FUNCTION Matrix_DeterminateSquare : BOOL
VAR_INPUT
	M : REFERENCE TO Matrix;
END_VAR
VAR_OUTPUT
	Res : LREAL;
END_VAR
VAR
	Sum : LREAL;
	Sign : LREAL;
	SubMatrix : ShrunkMatrixAccessor;
	
	Ci : UINT;
END_VAR

IF NOT(M.IsSquare) OR M.IsEmpty THEN
	Matrix_DeterminateSquare := FALSE;
	Res := 0;
	RETURN;
END_IF

Matrix_DeterminateSquare := TRUE;

IF M.Length = 1 THEN
	Res := M.GetRC(0,0);
ELSE
	Sum := 0;
	FOR Ci := 0 TO M.Cols-1 DO
		Sign := ((UINT_TO_INT(Ci)+1) MOD 2)*2 -1;//even columns are positive, odd columns are negative
		SubMatrix := M.GetShrunkMatrixAccessor(0,Ci);
		Sum := Sum + Sign * M.GetRC(0,Ci) * SubMatrix.GetDeterminant();//direct recursion is not accessible, but this should work
	END_FOR
	Res := Sum;
END_IF

END_FUNCTION

(* stored: Version 1.1.0.1, ProductVersion 3.1.4024.9
   POU Matrix_DeterminateSquare: Id {eb8e9d71-3179-0365-01f4-1666dd276213}, SpecialFunc None *)
